// TIA Portal V18 export
// export: Created 2025-12-01T12:39:35.5302033Z, ExportSetting None, DisplayName Totally Integrated Automation Portal, DisplayVersion V18 Update 5, DisplayName TIA Portal Openness, DisplayVersion V18 Update 5, DisplayName TIA Portal Teamcenter Gateway, DisplayVersion V18, DisplayName TIA Portal Version Control Interface, DisplayVersion V18, DisplayName STEP 7 Professional, DisplayVersion V18 Update 5, DisplayName STEP 7 Safety, DisplayVersion V18, DisplayName WinCC Professional, DisplayVersion V18 Update 5
VAR_GLOBAL   // PLC tag table "MES_NGCode"
END_VAR
VAR_GLOBAL CONSTANT   // user constants
   MES_NGCodeNG_Press : Int := 201;
   MES_NGCodeOK : Int := 0;
   MES_NGCodeIDIE : Int := 0;
   MES_NGCodeNG_illegal : Int := 201;
   MES_NGCodeNG_Manual : Int := 209;
END_VAR
